(* IEC 61131-3 sources: plc-home-automation/home_automation/lighting_heating_updated/src/watering, 3 files *)

(* ---- WateringGlobals.st ---- *)
VAR_GLOBAL CONSTANT
  C_WATERING_TIME_SLOTS : INT := 2;
END_VAR

VAR_GLOBAL

  // Global control
  WATERING_ENABLE : BOOL := TRUE;
  TEMPERATURE_BASED_WATERING_CONTROL   : BOOL := FALSE;
  RAIN_BASED_WATERING_CONTROL   : BOOL := TRUE;

  // Watering times
  WATERING_START_TIME       : ARRAY [1..C_WATERING_TIME_SLOTS] OF TIME;
  FRONT_GRASS_WATERING_TIME : ARRAY [1..C_WATERING_TIME_SLOTS] OF TIME;
  REAR_GRASS_WATERING_TIME  : ARRAY [1..C_WATERING_TIME_SLOTS] OF TIME;
  BUSHES_WATERING_TIME      : ARRAY [1..C_WATERING_TIME_SLOTS] OF TIME;

  FRONT_GRASS_START_TIME    : ARRAY [1..C_WATERING_TIME_SLOTS] OF TIME;
  FRONT_GRASS_END_TIME      : ARRAY [1..C_WATERING_TIME_SLOTS] OF TIME;
  REAR_GRASS_START_TIME     : ARRAY [1..C_WATERING_TIME_SLOTS] OF TIME;
  REAR_GRASS_END_TIME       : ARRAY [1..C_WATERING_TIME_SLOTS] OF TIME;
  BUSHES_START_TIME         : ARRAY [1..C_WATERING_TIME_SLOTS] OF TIME;
  BUSHES_END_TIME           : ARRAY [1..C_WATERING_TIME_SLOTS] OF TIME;

  FRONT_GRASS_WATERING_IN_PROGRESS : ARRAY [1..C_WATERING_TIME_SLOTS] OF BOOL;
  REAR_GRASS_WATERING_IN_PROGRESS : ARRAY [1..C_WATERING_TIME_SLOTS] OF BOOL;
  BUSHES_WATERING_IN_PROGRESS : ARRAY [1..C_WATERING_TIME_SLOTS] OF BOOL;

  // Temperature related control
  WATERING_CUTOFF_TEMPERATURE : REAL;
  FRONT_GRASS_WATERING_OFFSET : REAL;
  REAR_GRASS_WATERING_OFFSET  : REAL;
  FRONT_GRASS_WATERING_TEMPERATURE_COEFFICIENT : REAL;
  REAR_GRASS_WATERING_TEMPERATURE_COEFFICIENT  : REAL;

  // Waterting actuator controls
  FRONT_GRASS_WATERING_ON : BOOL := FALSE;
  REAR_GRASS_WATERING_ON : BOOL := FALSE;
  BUSHES_WATERING_ON : BOOL := FALSE;

END_VAR

(* ---- Watering.st ---- *)
PROGRAM WateringControl

  VAR_INPUT
  END_VAR
  VAR_OUTPUT
  END_VAR
  VAR
    rainEnabled : BOOL := TRUE;
    i : INT := 0;
  END_VAR
  VAR_TEMP
  END_VAR

  CURRENT_TIME := GetTime();
  rainEnabled := NOT (RAIN_BASED_WATERING_CONTROL AND RAIN_DETECTOR_IN);

  FOR i := 1 to C_WATERING_TIME_SLOTS DO

    IF TEMPERATURE_BASED_WATERING_CONTROL THEN
      FRONT_GRASS_WATERING_TIME[i] := REAL_TO_TIME((FRONT_GRASS_WATERING_OFFSET + FRONT_GRASS_WATERING_TEMPERATURE_COEFFICIENT * EXTERNAL_AVERAGE_TEMPERATURE) * 1000);
      REAR_GRASS_WATERING_TIME[i] := REAL_TO_TIME((REAR_GRASS_WATERING_OFFSET + REAR_GRASS_WATERING_TEMPERATURE_COEFFICIENT * EXTERNAL_AVERAGE_TEMPERATURE) * 1000);
      BUSHES_WATERING_TIME[i] := FRONT_GRASS_WATERING_TIME[i] + REAR_GRASS_WATERING_TIME[i];

      IF EXTERNAL_AVERAGE_TEMPERATURE < WATERING_CUTOFF_TEMPERATURE THEN
        FRONT_GRASS_WATERING_TIME[i] := T#00:00:00;
        REAR_GRASS_WATERING_TIME[i] := T#00:00:00;
        BUSHES_WATERING_TIME[i] := T#00:00:00;
      END_IF;

      IF FRONT_GRASS_WATERING_TIME[i] < T#00:00:00 THEN
        FRONT_GRASS_WATERING_TIME[i] := T#00:00:00;
      END_IF;
      IF REAR_GRASS_WATERING_TIME[i] < T#00:00:00 THEN
        REAR_GRASS_WATERING_TIME[i] := T#00:00:00;
      END_IF;
      IF BUSHES_WATERING_TIME[i] < T#00:00:00 THEN
        BUSHES_WATERING_TIME[i] := T#00:00:00;
      END_IF;
    END_IF;

    FRONT_GRASS_START_TIME[i] := WATERING_START_TIME[i];
    FRONT_GRASS_END_TIME[i]   := ADD_TIME(FRONT_GRASS_START_TIME[i], FRONT_GRASS_WATERING_TIME[i]);
    REAR_GRASS_START_TIME[i]  := FRONT_GRASS_END_TIME[i];
    REAR_GRASS_END_TIME[i]    := ADD_TIME(REAR_GRASS_START_TIME[i], REAR_GRASS_WATERING_TIME[i]);
    BUSHES_START_TIME[i]      := WATERING_START_TIME[i];
    BUSHES_END_TIME[i]        := ADD_TIME(BUSHES_START_TIME[i], BUSHES_WATERING_TIME[i]);

    // Start sections
    IF NOT FRONT_GRASS_WATERING_IN_PROGRESS[i] THEN
      IF CURRENT_TIME > FRONT_GRASS_START_TIME[i] THEN
        IF CURRENT_TIME < FRONT_GRASS_END_TIME[i] THEN
          FRONT_GRASS_WATERING_IN_PROGRESS[i] := TRUE;
          FRONT_GRASS_WATERING_ON := TRUE;
        END_IF;
      END_IF;
    END_IF;

    IF NOT REAR_GRASS_WATERING_IN_PROGRESS[i] THEN
      IF CURRENT_TIME > REAR_GRASS_START_TIME[i] THEN
        IF CURRENT_TIME < REAR_GRASS_END_TIME[i] THEN
          REAR_GRASS_WATERING_IN_PROGRESS[i] := TRUE;
          REAR_GRASS_WATERING_ON := TRUE;
        END_IF;
      END_IF;
    END_IF;

    IF NOT BUSHES_WATERING_IN_PROGRESS[i] THEN
      IF CURRENT_TIME > BUSHES_START_TIME[i] THEN
        IF CURRENT_TIME < BUSHES_END_TIME[i] THEN
          BUSHES_WATERING_IN_PROGRESS[i] := TRUE;
          BUSHES_WATERING_ON := TRUE;
        END_IF;
      END_IF;
    END_IF;

    // End sections

    IF FRONT_GRASS_WATERING_IN_PROGRESS[i] AND (CURRENT_TIME > FRONT_GRASS_END_TIME[i]) THEN
      FRONT_GRASS_WATERING_IN_PROGRESS[i] := FALSE;
      FRONT_GRASS_WATERING_ON := FALSE;
    END_IF;

    IF REAR_GRASS_WATERING_IN_PROGRESS[i] AND (CURRENT_TIME > REAR_GRASS_END_TIME[i]) THEN
      REAR_GRASS_WATERING_IN_PROGRESS[i] := FALSE;
      REAR_GRASS_WATERING_ON := FALSE;
    END_IF;

    IF BUSHES_WATERING_IN_PROGRESS[i] AND (CURRENT_TIME > BUSHES_END_TIME[i]) THEN
      BUSHES_WATERING_IN_PROGRESS[i] := FALSE;
      BUSHES_WATERING_ON := FALSE;
    END_IF;

  END_FOR;

  FRONT_GRASS_WATERING_ON := FRONT_GRASS_WATERING_ON AND WATERING_ENABLE AND rainEnabled;
  REAR_GRASS_WATERING_ON  := REAR_GRASS_WATERING_ON AND WATERING_ENABLE AND rainEnabled;
  BUSHES_WATERING_ON      := BUSHES_WATERING_ON AND WATERING_ENABLE AND rainEnabled;

  FRONT_GRASS_WATERING_OUT := FRONT_GRASS_WATERING_ON;
  REAR_GRASS_WATERING_OUT  := REAR_GRASS_WATERING_ON;
  BUSHES_WATERING_OUT      := BUSHES_WATERING_ON;

END_PROGRAM

(* ---- WateringInit.st ---- *)
PROGRAM WateringInit
  VAR_INPUT
  END_VAR
  VAR_OUTPUT
  END_VAR
  VAR
    initialised : BOOL := FALSE;
    i : INT := 0;
  END_VAR
  VAR_TEMP
  END_VAR

  WATERING_START_TIME[1]       := T#06:00:00;
  FRONT_GRASS_WATERING_TIME[1] := T#00:02:00;
  REAR_GRASS_WATERING_TIME[1]  := T#00:08:00;
  BUSHES_WATERING_TIME[1]       := T#00:08:00;

  FRONT_GRASS_START_TIME[1] := T#06:00:00;
  FRONT_GRASS_END_TIME[1]   := T#06:02:00;
  REAR_GRASS_START_TIME[1]  := T#06:02:00;
  REAR_GRASS_END_TIME[1]    := T#06:10:00;
  BUSHES_START_TIME[1]      := T#06:00:00;
  BUSHES_END_TIME[1]        := T#06:08:00;

  WATERING_START_TIME[2]       := T#20:00:00;
  FRONT_GRASS_WATERING_TIME[2] := T#00:01:00;
  REAR_GRASS_WATERING_TIME[2]  := T#00:04:00;
  BUSHES_WATERING_TIME[2]      := T#00:08:00;

  FRONT_GRASS_START_TIME[2] := T#20:00:00;
  FRONT_GRASS_END_TIME[2]   := T#20:01:00;
  REAR_GRASS_START_TIME[2]  := T#20:01:00;
  REAR_GRASS_END_TIME[2]    := T#20:05:00;
  BUSHES_START_TIME[2]      := T#20:00:00;
  BUSHES_END_TIME[2]        := T#20:08:00;

  FOR i := 1 to C_WATERING_TIME_SLOTS DO
    FRONT_GRASS_WATERING_IN_PROGRESS[i] := FALSE;
    REAR_GRASS_WATERING_IN_PROGRESS[i] := FALSE;
    BUSHES_WATERING_IN_PROGRESS[i] := FALSE;
  END_FOR;

  WATERING_CUTOFF_TEMPERATURE := 8;
  FRONT_GRASS_WATERING_OFFSET := 0;
  REAR_GRASS_WATERING_OFFSET  := 0;
  FRONT_GRASS_WATERING_TEMPERATURE_COEFFICIENT := 30;
  REAR_GRASS_WATERING_TEMPERATURE_COEFFICIENT  := 12;

  IF NOT initialised THEN
    initialised := TRUE;
  END_IF;

END_PROGRAM
